PROGRAM PRG_FB_CTRL_PID
VAR
	fSetpointValue					: LREAL;
	fActualValue					: LREAL;
	fManSyncValue					: LREAL;
	bSync							: BOOL;

	fOut							: LREAL;
	bHold							: BOOL;

	eMode							: E_CTRL_MODE;
	stCTRL_PID_PARAMS				: ST_CTRL_PID_PARAMS;
	stCTRL_PID_PARAMS_MTR_1			: ST_CTRL_PID_PARAMS;

	eErrorId						: E_CTRL_ERRORCODES;
	bError							: BOOL;
	bARWactive						: BOOL;

	(* controllers *)
	fbCTRL_PID						: FB_CTRL_PID;
	fbCTRL_PID_B28_MTR_1			: FB_CTRL_PID;

	bInit							: BOOL	:= TRUE;
	bInit_MTR_1						: BOOL	:= TRUE;
	fbTON							: TON;
	
	
	
	
END_VAR


IF CMD.Plant_B28_Control.PO_MODE = 2 THEN
	eMode :=  4;	
END_IF
IF CMD.Plant_B28_Control.PO_MODE = 1  THEN
	eMode :=  2;
ELSE
	eMode :=  0;	
END_IF


IF bInit THEN
	(* init parameter struct *)
	stCTRL_PID_PARAMS.tCtrlCycleTime		:= T#500MS;	//used to control the actual sample time of the PID algorythm, must be = or > than the task cycle time
	stCTRL_PID_PARAMS.tTaskCycleTime		:= T#100MS;		// must be the same as the cycletime configured in the task which the regulator is called in (CyclicTask100Ms)
	stCTRL_PID_PARAMS.fKp					:= 5.0;			(* proportional gain Kp				*)
	stCTRL_PID_PARAMS.tTn					:= T#100S;		(*  Tn								*)
	stCTRL_PID_PARAMS.tTv					:= T#200MS;		(*  Tv								*)
	stCTRL_PID_PARAMS.tTd					:= T#500MS;		(*  Td								*)
	stCTRL_PID_PARAMS.fOutMaxLimit			:=  100.0;			(* maximum output limit			(for  fillValve)	*) 
	stCTRL_PID_PARAMS.fOutMinLimit			:= -0.0;			(* minimum output limit			(for  fillValve)	*)

	(* set the mode to ACTIVE --> normal operation *)
	eMode := eCTRL_MODE_ACTIVE;

	(* reset the init flag *)
	bInit := FALSE;
END_IF

IF bInit_MTR_1 THEN
	(* init parameter struct *)
	stCTRL_PID_PARAMS_MTR_1.tCtrlCycleTime		:= T#500MS;	//used to control the actual sample time of the PID algorythm, must be = or > than the task cycle time
	stCTRL_PID_PARAMS_MTR_1.tTaskCycleTime		:= T#100MS;		// must be the same as the cycletime configured in the task which the regulator is called in (CyclicTask100Ms)
	stCTRL_PID_PARAMS_MTR_1.fKp					:= 0.1;			(* proportional gain Kp				*)
	stCTRL_PID_PARAMS_MTR_1.tTn					:= T#100S;		(*  Tn								*)
	stCTRL_PID_PARAMS_MTR_1.tTv					:= T#100MS;		(*  Tv								*)
	stCTRL_PID_PARAMS_MTR_1.tTd					:= T#500MS;		(*  Td								*)
	stCTRL_PID_PARAMS_MTR_1.fOutMaxLimit			:=  100.0;			(* maximum output limit			(for  fillValve)	*) 
	stCTRL_PID_PARAMS_MTR_1.fOutMinLimit			:= -0.0;			(* minimum output limit			(for  fillValve)	*)

	(* set the mode to ACTIVE --> normal operation *)
	eMode := eCTRL_MODE_ACTIVE;

	(* reset the init flag *)
	bInit_MTR_1 := FALSE;
END_IF

(*
TYPE E_CTRL_MODE :
(
    eCTRL_MODE_IDLE       := 0, (* mode idle *)
    eCTRL_MODE_PASSIVE    := 1, (* mode passive *)
    eCTRL_MODE_ACTIVE     := 2, (* mode active *)
    eCTRL_MODE_RESET      := 3, (* mode reset *)
    eCTRL_MODE_MANUAL     := 4, (* mode manual *)
    eCTRL_MODE_TUNE       := 5, (* mode tuning *)
    eCTRL_MODE_SELFTEST       := 6, (* mode selftest *)
    eCTRL_MODE_SYNC_MOVEMENT  := 7  (* mode synchronize *)
);
END_TYPE
*)

(*
fActualValue :=  FIO.iPV; 	//FIO.rLevelMeter;
fSetpointValue := FIO.iSP; //FIO.rSetPoint (0-10V Scaled to 0-300 cm)

(* copy var to scope var *)
GVL.fSetpointValueToScope 	:= fSetpointValue;
GVL.fActualValueToScope 	:= fActualValue;
*)

(* call controller *)
fbCTRL_PID(		fSetpointValue		:= fSetpointValue,
				fActualValue		:= fActualValue, //feedback value (proces variable)
				fManSyncValue		:= fManSyncValue, // controll fOut directly with 0-100 %?
				bSync				:= bSync,
				eMode				:= eMode,
				bHold				:= bHold,
				stParams			:= stCTRL_PID_PARAMS,
				fOut				=> fOut, // output to PID
				bARWactive			=> bARWactive,
				eErrorId			=> eErrorId,
				bError				=> bError
				);

(*
(* copy var to scope var *)
GVL.fOutToScope := fOut;
FIO.rFillValve :=  fOut;

GVL.outputDischargeValve := fOut;

(********************************************* CALL MOTOR 1 ***********************************************)
*)
fActualValue :=  HMI.outputFromPressure_1; 	// Fra tryk sensor (0-32767 --> 0-100)
fSetpointValue := PAR.MTR_1_SP; //F



fbCTRL_PID_B28_MTR_1(
				fSetpointValue		:= fSetpointValue,
				fActualValue		:= fActualValue, //feedback value (proces variable)
				fManSyncValue		:= fManSyncValue, // controll fOut directly with 0-100 %?
				bSync				:= bSync,
				eMode				:= eMode,
				bHold				:= bHold,
				stParams			:= stCTRL_PID_PARAMS_MTR_1,
				fOut				=> fOut, // output to PID
				bARWactive			=> bARWactive,
				eErrorId			=> eErrorId,
				bError				=> bError
				);

SIM.MTR_1_InputFromPID := LREAL_TO_DINT(fOut);

END_PROGRAM

(* stored: Version 1.1.0.1, ProductVersion 3.1.4024.13
   POU PRG_FB_CTRL_PID: Id {ab4b9d68-903a-4dd7-8d89-3218bcdb26f1}, SpecialFunc None *)
